// TIA Portal project "P1_Ejercicio2" (V15.1)

(* hardware
DEVICE "S7-1200 station_1"  S7-1200 Station
   slot 0: "Rack_0"  S7-1200 Rack  Rack  V1.0
   slot 1: "PLC_1"  CPU 1215C AC/DC/Rly  6ES7 215-1BG40-0XB0  V4.2
DEVICE "HMI_1"  KTP900 Basic PN
   slot 0: "HMI_1"  KTP900 Basic PN  6AV2 123-2JB03-0AX0  15.1.0.0
   slot 1: "HMI_RT_1"  KTP900 Basic PN  6AV2 123-2JB03-0AX0  15.1.0.0
   slot 5: "HMI_1.IE_CP_1"  PROFINET Interface  15.0.1.0
      slot 1: "Interfaz PROFINET_1"  PROFINET Interface
         slot 1: "Port_1"  Port
*)

// ===== PLC "PLC_1"  CPU 1215C AC/DC/Rly =====

VAR_GLOBAL   // PLC tag table "Tabla de variables estándar"
   "zona 1" AT %M0.0 : Bool;
   "zona 2" AT %M0.1 : Bool;
   "sistema alarma ON/OFF" AT %M0.2 : Bool;
   "alarma manual" AT %M0.3 : Bool;
   "LED sistema de alarma" AT %M10.0 : Bool;
   "Dispara sirena alarma" AT %M10.1 : Bool;
   "señal alerta baja" AT %M10.2 : Bool;
   "relé interface externo" AT %M10.3 : Bool;
   "temp 90s superado" AT %M20.0 : Bool;
   "temp 60s superado" AT %M20.1 : Bool;
END_VAR

// folder: System blocks/Program resources

DATA_BLOCK "Temporizador 90s"   // DB1
{ S7_Optimized_Access := 'TRUE' }
AUTHOR : Simatic
FAMILY : IEC
NAME : IEC_TMR
VERSION : 1.0
// stored: InstanceOfName IEC_TIMER
"IEC_TIMER"
BEGIN
END_DATA_BLOCK

DATA_BLOCK "Temporizador 60s"   // DB2
{ S7_Optimized_Access := 'TRUE' }
AUTHOR : Simatic
FAMILY : IEC
NAME : IEC_TMR
VERSION : 1.0
// stored: InstanceOfName IEC_TIMER
"IEC_TIMER"
BEGIN
END_DATA_BLOCK

// folder: (top level)

ORGANIZATION_BLOCK "Main"   // OB1, LAD, ProgramCycle
TITLE = "Main Program Sweep (Cycle)" / Ejercicio 2
{ S7_Optimized_Access := 'TRUE' }
VERSION : 0.1
   VAR_INPUT
      Initial_Call : Bool;   // Initial call of this OB
      Remanence : Bool;   // =True, if remanent data are available
   END_VAR
BEGIN

REGION Network 1
   // ⚈Si el sistema no está activado, el LED (%M10.0) parpadea al estar abiertas la zona 1 (%M0.0) o 2 (%M0.1).
   // ⚈La entrada 1 (%M0.0) vigila la zona 1 (entrada delantera, sala de estar, cocina y dormitorio 3).
   // Entrada normalmente cerrada. (Abierto=”0”, Cerrado=”1”).
   // ⚈La entrada 2 (%M0.1) vigila la zona 2 (dormitorio 1, dormitorio 2, baño y entrada trasera).
   // Entrada normalmente cerrada. (Abierto=”0”, Cerrado=”1”).
   // ⚈La salida 1 (%M10.0) controla el LED del sistema de alarma. Estará encendido si está activado y parpadeante si está desactivado, estando abiertas la zona 1 o la zona 2.
   // ⚈Si el sistema está activado (girando la llave a la posición “on”, lo que activa la entrada %M0.2),
   // el programa arranca un temporizador de retardo de 90 segundos para que el propietario
   // pueda salir de la vivienda. Durante ese tiempo de retardo, el programa no reacciona si se abre
   // alguna de las zonas (%M0.0 ó %M0.1).
   // ⚈Una vez arrancada la secuencia de notificación, si se desactiva el sistema (girando la llave a la posición “off”, lo que desactiva %M0.2), el programa pone a ”0” las salidas (%M10.0 y %M10.2) y los temporizadores.
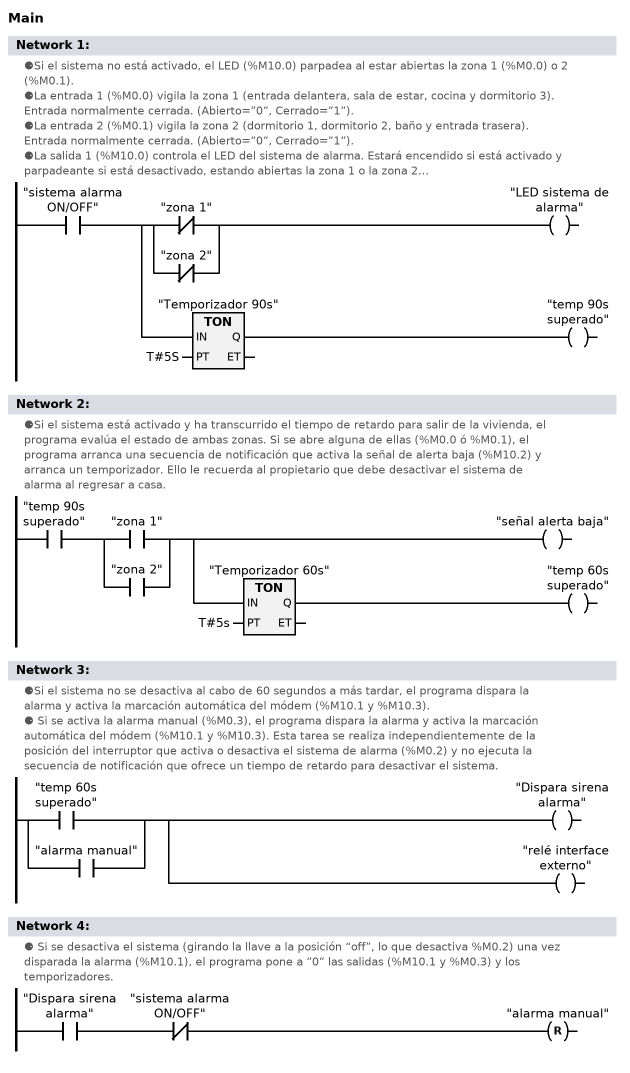
   "LED sistema de alarma" := "sistema alarma ON/OFF" AND (NOT "zona 1" OR NOT "zona 2");
   "Temporizador 90s".TON(IN := "sistema alarma ON/OFF", PT := T#5S);
   "temp 90s superado" := "Temporizador 90s".Q;
END_REGION

REGION Network 2
   // ⚈Si el sistema está activado y ha transcurrido el tiempo de retardo para salir de la vivienda, el
   // programa evalúa el estado de ambas zonas. Si se abre alguna de ellas (%M0.0 ó %M0.1), el
   // programa arranca una secuencia de notificación que activa la señal de alerta baja (%M10.2) y
   // arranca un temporizador. Ello le recuerda al propietario que debe desactivar el sistema de
   // alarma al regresar a casa.
   "señal alerta baja" := "temp 90s superado" AND ("zona 1" OR "zona 2");
   "Temporizador 60s".TON(IN := "señal alerta baja", PT := T#5s);
   "temp 60s superado" := "Temporizador 60s".Q;
END_REGION

REGION Network 3
   // ⚈Si el sistema no se desactiva al cabo de 60 segundos a más tardar, el programa dispara la
   // alarma y activa la marcación automática del módem (%M10.1 y %M10.3).
   // 
   // ⚈ Si se activa la alarma manual (%M0.3), el programa dispara la alarma y activa la marcación
   // automática del módem (%M10.1 y %M10.3). Esta tarea se realiza independientemente de la
   // posición del interruptor que activa o desactiva el sistema de alarma (%M0.2) y no ejecuta la
   // secuencia de notificación que ofrece un tiempo de retardo para desactivar el sistema.
   RUNG wire#powerrail
      Contact( "temp 60s superado" )
      wire#w1
      Coil( "Dispara sirena alarma" )
   END_RUNG
   RUNG wire#powerrail
      Contact( "alarma manual" )
   END_RUNG wire#w1
   RUNG wire#w1
      Coil( "relé interface externo" )
   END_RUNG
   // the same network as SCL:
   "Dispara sirena alarma" := "temp 60s superado" OR "alarma manual";
   "relé interface externo" := "Dispara sirena alarma";
END_REGION

REGION Network 4
   // ⚈ Si se desactiva el sistema (girando la llave a la posición “off”, lo que desactiva %M0.2) una vez
   // disparada la alarma (%M10.1), el programa pone a ”0” las salidas (%M10.1 y %M0.3) y los
   // temporizadores.
   RUNG wire#powerrail
      Contact( "Dispara sirena alarma" )
      I_Contact( "sistema alarma ON/OFF" )
      R_Coil( "alarma manual" )
   END_RUNG
   // the same network as SCL:
   IF "Dispara sirena alarma" AND NOT "sistema alarma ON/OFF" THEN "alarma manual" := FALSE; END_IF;
END_REGION
END_ORGANIZATION_BLOCK

(* ===== HMI "HMI_RT_1" =====
system functions are stored by id; their names below are inferred from use
connection "HMI_Conexión_1": ETHERNET, SMART_S7_1200_OMS

HMI tags "Tabla de variables estándar"
   "Número_imagen_variable" : UInt, internal
   "sistema alarma ON/OFF" : Bool = PLC "sistema alarma ON/OFF" AT %M0.2, 1 s
   "LED sistema de alarma" : Bool = PLC "LED sistema de alarma" AT %M10.0, 1 s
   "Dispara sirena alarma" : Bool = PLC "Dispara sirena alarma" AT %M10.1, 1 s
   "zona 1" : Bool = PLC "zona 1" AT %M0.0, 1 s
   "zona 2" : Bool = PLC "zona 2" AT %M0.1, 1 s
   "temp 90s superado" : Bool = PLC "temp 90s superado" AT %M20.0, 1 s
   "temp 60s superado" : Bool = PLC "temp 60s superado" AT %M20.1, 1 s
   "alarma manual" : Bool = PLC "alarma manual" AT %M0.3, 1 s

text list "Nombre_imagen_lista_texto": 1 'Imagen raíz'

Template "Plantilla_1" 800x480
   Button "Salir" at 722,440 size 55x39; TextOff 'Salir'; PictureOff "ExitRuntime_KTP900_Basic_PN_TR"; PictureOn "ExitRuntime_KTP900_Basic_PN_TR"
      on Release: StopRuntime(0)
   Button "Template_Button" at 622,440 size 55x39; TextOff 'Text'
   Button "Template_Button_1" at 522,440 size 55x39; TextOff 'Text'
   Button "Template_Button_2" at 422,440 size 55x39; TextOff 'Text'
   Button "Template_Button_3" at 322,440 size 55x39; TextOff 'Text'
   Button "Template_Button_4" at 222,440 size 55x39; TextOff 'Text'
   Button "Avisos" at 122,440 size 55x39; TextOff 'Avisos'; PictureOff "AlarmDisplay_KTP900_Basic_PN_TR"; PictureOn "AlarmDisplay_KTP900_Basic_PN_TR"
      on Release: function_ef3f5d25("Ventana de avisos_no_acusado", -1)
   Button "Imagen inicial" at 22,440 size 55x39; TextOff 'Imagen inicial'; PictureOff "NavigateHome_KTP900_Basic_PN_TR"; PictureOn "NavigateHome_KTP900_Basic_PN_TR"
      on Release: ActivateScreen("Imagen raíz", 0)
   SymbolicIOField "Imagen_campo_ES_simbólico" at 73,7 size 620x26; TextOff '0'; TextOn '1'; TextList "Nombre_imagen_lista_texto"
      ProcessValue <- "Número_imagen_variable"
      on Change: ActivateScreenByNumber("Número_imagen_variable", 0)
   DateTimeField "HmiScreenItemData" at 695,20 size 105x20
   DateTimeField "HmiScreenItemData_1" at 695,0 size 105x20
   GraphicView "Logotipo" at 0,0 size 71x40; Picture "Logotipo de HMI_1"

screen "Imagen raíz" 800x480, template "Plantilla_1"
   on GenerateScreen: SetTag("Número_imagen_variable", 1)
   Switch "Interruptor_1" at 49,75 size 64x32; CaptionText 'Switch'; TextOff 'OFF'; TextOn 'ON'
      ProcessValue <- "sistema alarma ON/OFF"
   Circle "Círculo_1" at 378,84 size 48x48
      Appearance <- "LED sistema de alarma"
   TextField "Campo de texto_2" at 10,52 size 153x20; Text 'sistema alarma ON/OFF'
   TextField "Campo de texto_1" at 325,61 size 150x20; Text 'LED sistema de alarma'
   TextField "Campo de texto_3" at 426,90 size 128x15; Text 'Parpadeo = desactivado'
   TextField "Campo de texto_4" at 426,105 size 113x15; Text 'Encendido = activado'
   Circle "Círculo_2" at 375,208 size 48x48
      Appearance <- "Dispara sirena alarma"
   TextField "Campo de texto_5" at 375,188 size 52x20; Text 'SIRENA'
   TextField "Campo de texto_6" at 421,215 size 66x15; Text 'Verde = ON'
   TextField "Campo de texto_7" at 423,230 size 64x15; Text 'Rojo = OFF'
   Switch "Interruptor_2" at 57,253 size 64x32; TextOn 'ON'; CaptionText 'Switch'; TextOff 'OFF'
      ProcessValue <- "alarma manual"
   TextField "Campo de texto_8" at 19,236 size 151x20; Text 'Alarma Manual ON/OFF'
   Rectangle "Rectángulo_1" at 219,71 size 53x32
      Appearance <- "zona 1"
   Rectangle "Rectángulo_2" at 219,130 size 52x34
      Appearance <- "zona 2"
   TextField "Campo de texto_9" at 224,51 size 48x20; Text 'Zona 1'
   TextField "Campo de texto_10" at 219,110 size 48x20; Text 'Zona 2'
   Line "Línea_1" at 112,84 size 107x5
      Appearance <- "sistema alarma ON/OFF"
   Ellipse "Elipse_1" at 57,182 size 56x34
      Appearance <- "temp 90s superado"
   Ellipse "Elipse_2" at 219,194 size 56x34
      Appearance <- "temp 60s superado"
   TextField "Campo de texto_11" at 50,163 size 66x20; Text 'Temp 90s'
   TextField "Campo de texto_12" at 213,175 size 66x20; Text 'Temp 60s'
   Line "Línea_3" at 106,94 size 113x55
      Appearance <- "sistema alarma ON/OFF"
*)